(* CODESYS project WagoApp_1.11.0.x_Cloud_FbCollectionLogger_Example_03.ecp

Project tree, tasks and I/O mapping:
  PFC_KQL : 750-8210 PFC200 G2 4ETH, WAGO, order no. 0750-8210, version 5.17.3.3
    application Application
      libraries: ; WagoAppCloud, * (WAGO); WagoAppTime, 1.7.3.5 (WAGO); WagoAppControlSuite, 1.0.2.0 (WAGO)
      task PLC_Task (cyclic, interval 50 ms, priority 14) calls Prg_To_Cloud
      program Prg_To_Cloud [ST]
      trace Trace (task PLC_Task): Prg_To_Cloud.rSineP, Prg_To_Cloud.rValue
      FbOnChange/
        function block FbChangeOfValue_Bool [ST]
        function block FbChangeOfValue_Byte [ST]
        function block FbChangeOfValue_Dword [ST]
        function block FbChangeOfValue_Real [ST]
    ProjectConfiguration
    Kbus : Kbus, WAGO, version 1.4.0.2
        unmapped channels: K-BUS diagnostics
      _16_DO_Generic : 075x-16DO, WAGO, order no. 075x-16DO, version 0.0.0.13
          settings: K-BUS Module slot index = 3
          output wOut : WORD  // _OUT
      _2_DO_Generic : 075x-2DO, WAGO, order no. 075x-2DO, version 0.0.0.13
          settings: K-BUS Module slot index = 1
          output xCloudConnected : BOOL  // _OUT._OUT
          output xCloudError : BOOL  // _OUT._OUT
          unmapped channels: _OUT
      _16_DI_Generic : 075x-16DI, WAGO, order no. 075x-16DI, version 0.0.0.13
          settings: K-BUS Module slot index = 2
          input  wIn : WORD  // _IN
      _2AI_0_10_VDC_SE : 0750-0467, WAGO, order no. 0750-0467, version 0.0.0.9
          settings: K-BUS Module slot index = 4
          input  wAnalog_0_10V_1 : WORD  // _IW 1
          input  wAnalog_0_10V_2 : WORD  // _IW 2
      _2AI_TC_K_Diagn_Adjust : 0750-0469/0003-0000, WAGO, order no. 0750-0469/0003-0000, version 0.0.0.9
          settings: K-BUS Module slot index = 5
          input  iThermo1 : INT  // _IINT 1
          input  iThermo2 : INT  // _IINT 2
      _2AO_0_10_VDC : 0750-0550, WAGO, order no. 0750-0550, version 0.0.0.9
          settings: K-BUS Module slot index = 6
          output wAnalogOut_0_10V_1 : WORD  // _QW 1
          output wAnalogOut_0_10V_2 : WORD  // _QW 2
    MODBUS
      MODBUS : MODBUS, WAGO, order no. n/a, version 1.1.1.16
    Common.PCI
    EtherNet/IP
      Ethernet : Ethernet, WAGO, version 35.17.0.0
          settings: IPAddress = [192, 168, 1, 103]; SubnetMask = [0, 0, 0, 0]; MACAddress = [16#00, 16#00, 16#00, 16#00, 16#00, 16#00]; NetworkInterfaceName = 'br0'; NetworkInterfaceName = "br0"
  EC_PIO3_C : Edge Controller PIO3, WAGO, order no. 0752-8303, version 5.17.3.3
    application Application
      libraries: ; WagoAppTime, 1.7.3.5 (WAGO)
      task PLC_Task (cyclic, interval t#50ms, priority 15) calls PLC_PRG
      program PLC_PRG [ST]
    MODBUS
      MODBUS : MODBUS, WAGO, order no. n/a, version 1.1.1.16
    CANbus
    TP600_Onboard_IO : TP600 Onboard IO, WAGO, version 0.0.1.2
        output bOut : BYTE  // _OUT
        unmapped channels: _IN
    Common.PCI
    EtherNet/IP
      Ethernet : Ethernet, WAGO, version 35.17.0.0
          settings: IPAddress = [192, 168, 1, 14]; SubnetMask = [0, 0, 0, 0]; MACAddress = [16#00, 16#00, 16#00, 16#00, 16#00, 16#00]; NetworkInterfaceName = 'br0'; NetworkInterfaceName = "br0"
    Serial
      COM1 : COM1, WAGO, version 0.0.0.19
  00000000-0000-0000-0000-000000000000|C:\Users\Admin\AppData\Local\Temp\6c95a57c3216420fa36a3ac6dc2d92b7\e868b832187f4f1a859da50215710801\20221104120952\Project.xml
*)

// PFC_KQL/Application/Prg_To_Cloud
(* Purpose of the example program: 
	FbCollectionLogger will sample 3 collections in different modes.
	- Collection 1: EQUALLY_SPACED_COLLECTION_SAMPLES
	- Collection 2: UNEQUALLY_SPACED_CUSTOMIZED_SAMPLES
	- Collection 3: LIBRARY_DEFAULT_AUTOMATIC
*)
PROGRAM Prg_To_Cloud
VAR RETAIN
	(* Remanent variables *)
	tSampleInterval1 : TIME := T#10s;
	tPublishInterval1 : TIME := T#20S;
	tPublishInterval2 : TIME := T#20S;
	tSampleInterval3 : TIME := T#60S;
	tPublishInterval3 : TIME := T#120S;
xEnablePID: BOOL;rKp: REAL := 1.4;rTn: REAL := 19.89;rTv: REAL := 0.021;END_VAR

VAR
	

	(* Define three collections*)
	aCollections: ARRAY[0..2] OF WagoAppCloud.typCollection;

	(* Define the variables for the collections*)
	aVariableDescriptions1: ARRAY[0..3] OF WagoAppCloud.typVariableDescription;
	aVariableDescriptions2: ARRAY[0..2] OF WagoAppCloud.typVariableDescription;
	aVariableDescriptions3: ARRAY[0..5] OF WagoAppCloud.typVariableDescription;
	
	oFbCollectionLogger: WagoAppCloud.FbCollectionLogger;
	
	(* Timer *)
	xEnableTimer: BOOL := TRUE;
	tCyclicTimerSendTagCollection: TON;

	oFbChangeOfValue_Dword: FbChangeOfValue_Dword;	
	
	rPercentage1: REAL;
	rPercentage2: REAL;
	rTemperature1: REAL;
	rTemperature2: REAL;

	oFbChangeOfValue: FbChangeOfValue_Bool;
	xInputChanged: BOOL;
	xOutputChanged: BOOL;
	x: REAL := 0.01;
	wValue: WORD;
	rSineP: REAL;
	rValue: REAL;
	oFbStatus_WagoProtocol: WagoAppCloud.FbStatus_WagoProtocol;
	rCache: REAL;
	tSampleInterval1_10Minute: TIME := t#10m;
	xOutSend: BOOL;
	oFbChangeOfValue2: FbChangeOfValue_Bool;
	typComp: WagoAppTime.WagoTypes.typWagoTimeComponents;
	oRT: R_TRIG;
	
	oFb_PID_01: WagoAppControlSuite.Fb_PID_01;
	
	rSetpointTemperature1: REAL := 36.4;
	tSampleRate: TIME := T#100ms;
	
	
	
	rOutputMax: REAL := 100;
	rOutputMin: REAL := 0;
	xManualOperation: BOOL;
	rManualValue: REAL := 42.42;
	typConfiguration: WagoAppControlSuite.typPID_Configuration;
	rY: REAL;
	xLimitReached: BOOL;
	xLimitMaxReached: BOOL;
	xLimitMinReached: BOOL;
	tPublishInterval_USCD: TIME := T#10m;
	oFbChangeOfValue_Real: ARRAY[1..4] OF FbChangeOfValue_Real;
	oFbChangeOfValue_Bool_PID1,oFbChangeOfValue_Bool_PID2 :FbChangeOfValue_Bool;
END_VAR


typComp:=WagoAppTime.FuGetLocalTimeComponents();
oRT(CLK:=typComp.uiSecond.0);
IF oRT.Q THEN
	
	
	rPercentage1:= IoConfig_Globals_Mapping.wAnalog_0_10V_1/327.6;
	rPercentage2:= IoConfig_Globals_Mapping.wAnalog_0_10V_2/327.6;
	
	rTemperature1:= IoConfig_Globals_Mapping.iThermo1/10.0;
	rTemperature2:= IoConfig_Globals_Mapping.iThermo2/10.0;
	
	IF x > 3.14 THEN
		x:=0;
		ELSE 
			x:=x+0.01;	
	END_IF
	rSineP:=SIN(x);
	rValue:=rSineP * 32760;
	wValue:=TO_WORD(rValue);
END_IF

oFb_PID_01(
	xEnable:= 		xEnablePID, 
	rActualValue:=	rTemperature1 , 
	rSetpointValue:=rSetpointTemperature1 , 
	tSampleRate:= 	tSampleRate, 
	rKp:=	rKp , 
	rTn:= 	rTn, 
	rTv:=	rTv , 
	rOutputMax:=		rOutputMax, 
	rOutputMin:=		rOutputMin , 
	xManualOperation:= xManualOperation, 
	rManualValue:= 		rManualValue, 
	typConfiguration:= 	typConfiguration, 
	rY=> rY, 
	xLimitReached=>   xLimitReached , 
	xLimitMaxReached=>xLimitMaxReached , 
	xLimitMinReached=>xLimitMinReached);
//Generate some values for AO and DO	
IoConfig_Globals_Mapping.wAnalogOut_0_10V_1:= wValue;
IoConfig_Globals_Mapping.wOut:=(IoConfig_Globals_Mapping.wAnalog_0_10V_1 + IoConfig_Globals_Mapping.wAnalog_0_10V_2)/2;

(* Configuration of the collections and variables *)
	(* Init collection 1 *)
	aVariableDescriptions1[0].pAddress := ADR(rPercentage1);
	aVariableDescriptions1[0].eValueType := WagoAppCloud.VVT_REAL;
	aVariableDescriptions1[0].dwTypeId := 1;
	aVariableDescriptions1[0].sTag := 'Inflow1';
	aVariableDescriptions1[0].sUnit := '';
	
	aVariableDescriptions1[1].pAddress := ADR(rPercentage2);
	aVariableDescriptions1[1].eValueType := WagoAppCloud.VVT_REAL;
	aVariableDescriptions1[1].dwTypeId := 2;
	aVariableDescriptions1[1].sTag := 'Inflow2';
	aVariableDescriptions1[1].sUnit := '';
	
	aVariableDescriptions1[2].pAddress := ADR(rTemperature1);
	aVariableDescriptions1[2].eValueType := WagoAppCloud.VVT_REAL;
	aVariableDescriptions1[2].dwTypeId := 3;
	aVariableDescriptions1[2].sTag := 'Temperature1';
	aVariableDescriptions1[2].sUnit := '°C';
	
	aVariableDescriptions1[3].pAddress := ADR(rTemperature2);
	aVariableDescriptions1[3].eValueType := WagoAppCloud.VVT_REAL;
	aVariableDescriptions1[3].dwTypeId := 4;
	aVariableDescriptions1[3].sTag := 'Temperature2';
	aVariableDescriptions1[3].sUnit := '°C';
	
	
	(* Configuration of the collection. *)
	aCollections[0].dwCollectionId := 1;
	aCollections[0].sName := 'CollectionAnalogs';
	aCollections[0].pVariableDescriptions := ADR(aVariableDescriptions1);
	aCollections[0].dwVariablesCount := 4;
	(* Configuration of the mode to sampling the data. 
	In this case all variables of collection 1 will be send in equally spaced to the cloud. 
	The Trigger of a sample is set manual with the CollectionTrigger. *)
	aCollections[0].eSamplingDataMode := eSamplingMode.LIBRARY_DEFAULT_AUTOMATIC;
	aCollections[0].pSampleInterval := ADR(tSampleInterval1);
	aCollections[0].pPublishInterval := ADR(tPublishInterval1);
	
	(* Init collection 2 *)
	aVariableDescriptions2[0].pAddress := ADR(IoConfig_Globals_Mapping.wIn);
	aVariableDescriptions2[0].eValueType := WagoAppCloud.VVT_WORD;
	aVariableDescriptions2[0].dwTypeId := 1;
	aVariableDescriptions2[0].sTag := 'DI';
	aVariableDescriptions2[0].sUnit := 'Bin';
	
	aVariableDescriptions2[1].pAddress := ADR(IoConfig_Globals_Mapping.wOut);
	aVariableDescriptions2[1].eValueType := WagoAppCloud.VVT_WORD;
	aVariableDescriptions2[1].dwTypeId := 2;
	aVariableDescriptions2[1].sTag := 'DO';
	aVariableDescriptions2[1].sUnit := 'Bin';
	
	
	(* Configuration of the collection. *)
	aCollections[1].dwCollectionId := 2;
	aCollections[1].sName := 'CollectionDigital';
	aCollections[1].pVariableDescriptions := ADR(aVariableDescriptions2);
	aCollections[1].dwVariablesCount := 2;
	(* Configuration of the mode to sampling the data. 
	In this case at least one variable of collection 2 will be send irregularly to the cloud. 
	The Trigger of a sample is set manual with the CollectionTrigger or the VariableTrigger. *)
	aCollections[1].eSamplingDataMode := eSamplingMode.EQUALLY_SPACED_CUSTOMIZED_SAMPLES;
	aCollections[1].pPublishInterval := ADR(tPublishInterval2);
	(* Configuration of the collection. *)
	
	
	aVariableDescriptions3[0].pAddress := ADR(xEnablePID);
	aVariableDescriptions3[0].eValueType := WagoAppCloud.VVT_BOOL;
	aVariableDescriptions3[0].dwTypeId := 1;
	aVariableDescriptions3[0].sTag := 'EN';
	aVariableDescriptions3[0].sUnit := 'Bin';
	                     
	aVariableDescriptions3[1].pAddress := ADR(rSetpointTemperature1);
	aVariableDescriptions3[1].eValueType := WagoAppCloud.VVT_REAL;
	aVariableDescriptions3[1].dwTypeId := 2;
	aVariableDescriptions3[1].sTag := 'Setpoint';
	aVariableDescriptions3[1].sUnit := '°C';
	
	aVariableDescriptions3[2].pAddress := ADR(rKp);
	aVariableDescriptions3[2].eValueType := WagoAppCloud.VVT_REAL;
	aVariableDescriptions3[2].dwTypeId := 3;
	aVariableDescriptions3[2].sTag := 'P';
	aVariableDescriptions3[2].sUnit := '';
	                     
	aVariableDescriptions3[3].pAddress := ADR(rTn);
	aVariableDescriptions3[3].eValueType := WagoAppCloud.VVT_REAL;
	aVariableDescriptions3[3].dwTypeId := 4;
	aVariableDescriptions3[3].sTag := 'I';
	aVariableDescriptions3[3].sUnit := '';
	
	aVariableDescriptions3[4].pAddress := ADR(rTv);
	aVariableDescriptions3[4].eValueType := WagoAppCloud.VVT_REAL;
	aVariableDescriptions3[4].dwTypeId := 5;
	aVariableDescriptions3[4].sTag := 'D';
	aVariableDescriptions3[4].sUnit := '';
	                     
	aVariableDescriptions3[5].pAddress := ADR(xManualOperation);
	aVariableDescriptions3[5].eValueType := WagoAppCloud.VVT_BOOL;
	aVariableDescriptions3[5].dwTypeId := 6;
	aVariableDescriptions3[5].sTag := 'ManuelOperation';
	aVariableDescriptions3[5].sUnit := 'Bin';
	
	aCollections[2].dwCollectionId := 3;
	aCollections[2].sName := 'CollectionPID';
	aCollections[2].pVariableDescriptions := ADR(aVariableDescriptions3);
	aCollections[2].dwVariablesCount := 6;
	aCollections[2].eSamplingDataMode := eSamplingMode.UNEQUALLY_SPACED_CUSTOMIZED_SAMPLES;
	aCollections[2].pPublishInterval := ADR(tPublishInterval_USCD);
	
	
		
// BOOL on change
oFbChangeOfValue_Bool_PID1(xVariable:=xEnablePID 		, xTrigger:= aVariableDescriptions3[0].xVariableTrigger);
oFbChangeOfValue_Bool_PID2(xVariable:=xManualOperation  , xTrigger:= aVariableDescriptions3[5].xVariableTrigger);
 //xEnable PID Controller
 //Manuel Operation


// REAL  on change	
oFbChangeOfValue_Real[1](rInput:=rSetpointTemperature1 ,
						 rActivate:= 100 , 
						 rDeactivate:= 0, 							xTrigger:=aVariableDescriptions3[1].xVariableTrigger);
						 
oFbChangeOfValue_Real[2](rInput:=rKp , rActivate:=0 , rDeactivate:=100, xTrigger:=aVariableDescriptions3[2].xVariableTrigger);
oFbChangeOfValue_Real[3](rInput:=rTn , rActivate:=0 , rDeactivate:=100 ,xTrigger:=aVariableDescriptions3[3].xVariableTrigger);
oFbChangeOfValue_Real[4](rInput:=rTv , rActivate:=0 , rDeactivate:=100 ,xTrigger:=aVariableDescriptions3[4].xVariableTrigger);






(* Example to set the event if variable value exceeded the threshold values - Variable Trigger*)

oFbChangeOfValue(xVariable:=	wIn.0 OR 
								wIn.1 OR 
								wIn.2 OR 
								wIn.3 OR 
								wIn.4 OR 
								wIn.5 OR 
								wIn.6 OR 
								wIn.7, 
					xTrigger:= aVariableDescriptions2[0].xVariableTrigger);
	
oFbChangeOfValue2(xVariable:=	wOut.0 OR 
								wOut.1 OR 
								wOut.2 OR 
								wOut.3 OR 
								wOut.4 OR 
								wOut.5 OR 
								wOut.6 OR 
								wOut.7, 
					xTrigger:= aVariableDescriptions2[1].xVariableTrigger);

	
	

(* Example to set the event with a timer intervall - CollectionTrigger or VariableTrigger *)
	(* Set an event with an Timer to send the variables in an intervall to the cloud *)
	tCyclicTimerSendTagCollection(IN:= xEnableTimer, PT:= tSampleInterval1_10Minute);
	IF tCyclicTimerSendTagCollection.Q THEN
		aCollections[1].xCollectionTrigger := TRUE;
		aCollections[2].xCollectionTrigger:=TRUE;
		xEnableTimer := FALSE;
	ELSE
		xEnableTimer := TRUE;
	END_IF

	
oFbCollectionLogger(pCollections := ADR(aCollections), dwCollectionsCount := 3);
oFbStatus_WagoProtocol(
	xEnabled:=TRUE , 
	xError=>IoConfig_Globals_Mapping.xCloudError , 
	xCloudConnected=> IoConfig_Globals_Mapping.xCloudConnected, 
	rCacheFillLevel=> rCache , 
	xTelemetryDataTransmission=> , 
	bCollectionCounter=> , 
	uliOutgoingDataBlocks=> , 
	ErrorInformation=> , 
	oStatus=> );

END_PROGRAM

// PFC_KQL/Application/FbOnChange/FbChangeOfValue_Dword
(* The function block FbChangeOfValue_Dword shows an example how an event of a dword variable could be triggered.*)

FUNCTION_BLOCK FbChangeOfValue_Dword

VAR_INPUT
	dwInput 	: DWORD;
	dwActivate 	: DWORD;
	dwDeactivate : DWORD;
END_VAR

VAR_IN_OUT
	xTrigger	: BOOL;
END_VAR

VAR
	xLastSendedState: BOOL := FALSE;
END_VAR

(* Do only something when the VariableTrigger isn't activated (the VariableTrigger will be reset by the function block FbCollectionLogger) *)
IF NOT xTrigger THEN
	(* Two variations are to be considered during the analysis of the input values *)
	
	(* case 1: the activate threshold is greater as the deactivate threshold *)	
	IF dwActivate > dwDeactivate THEN
		(* rising edge *)
		IF (dwInput >= dwActivate) AND NOT xLastSendedState THEN
			xTrigger := TRUE;
			xLastSendedState := TRUE;
		(* falling edge *)
		ELSIF (dwInput <= dwDeactivate) AND xLastSendedState THEN
			xTrigger := TRUE;
			xLastSendedState := FALSE;
		END_IF
		
	(* case 2: the deactivate threshold is greater as the activate threshold *)
	ELSE
		(* rising edge *)
		IF (dwInput <= dwActivate) AND NOT xLastSendedState THEN
			xTrigger := TRUE;
			xLastSendedState := TRUE;(* save that the trigger after the rising edge is already set so that the trigger will be only set once *)
		(* falling edge *)
		ELSIF (dwInput >= dwDeactivate) AND xLastSendedState THEN
			xTrigger := TRUE;
			xLastSendedState := FALSE;
		END_IF
	END_IF
END_IF

END_FUNCTION_BLOCK

// PFC_KQL/Application/FbOnChange/FbChangeOfValue_Bool
FUNCTION_BLOCK FbChangeOfValue_Bool
VAR_INPUT
	xVariable : BOOL; 	(* Input value *)
END_VAR
VAR_IN_OUT
	xTrigger : BOOL; 	(* Variable Trigger - trigger is set only once when the value was changed and reset with the function block WagoAppCloud.FbCollectionLogger *)
END_VAR
VAR
	xLastSendedState : BOOL := FALSE; 	(* save the old value when this value was sending to the cloud to the if the value was changing *)
END_VAR

IF NOT xTrigger THEN
	IF NOT (xVariable = xLastSendedState) THEN
		xTrigger := TRUE;
		xLastSendedState := xVariable;
	END_IF
END_IF

END_FUNCTION_BLOCK

// PFC_KQL/Application/FbOnChange/FbChangeOfValue_Real
(* The function block FbChangeOfValue_Real shows an example how an event of a real variable could be triggered.
*)

FUNCTION_BLOCK FbChangeOfValue_Real

VAR_INPUT
	rInput 		: REAL;
	rActivate 	: REAL;
	rDeactivate : REAL;
END_VAR

VAR_IN_OUT
	xTrigger	: BOOL;
END_VAR

VAR
	xLastSendedState : BOOL := FALSE;
END_VAR

IF NOT xTrigger THEN
	IF rActivate > rDeactivate THEN
		IF (rInput >= rActivate) AND NOT xLastSendedState THEN
			xTrigger := TRUE;
			xLastSendedState := TRUE;
		ELSIF (rInput <= rDeactivate) AND xLastSendedState THEN
			xTrigger := TRUE;
			xLastSendedState := FALSE;
		END_IF
	ELSE
		IF (rInput <= rActivate) AND NOT xLastSendedState THEN
			xTrigger := TRUE;
			xLastSendedState := TRUE;
		ELSIF (rInput >= rDeactivate) AND xLastSendedState THEN
			xTrigger := TRUE;
			xLastSendedState := FALSE;
		END_IF
	END_IF
END_IF

END_FUNCTION_BLOCK

// EC_PIO3_C/Application/PLC_PRG
PROGRAM PLC_PRG
VAR
	typComp: WagoAppTime.WagoTypes.typWagoTimeComponents;
	oRT: R_TRIG;
END_VAR

typComp:=WagoAppTime.FuGetLocalTimeComponents();
oRT(CLK:=typComp.uiSecond.0);
IF oRT.Q THEN
	IF IoConfig_Globals_Mapping.bOut <=255 THEN
	IoConfig_Globals_Mapping.bOut:=IoConfig_Globals_Mapping.bOut+1;
	ELSE
		IoConfig_Globals_Mapping.bOut:=0;
	END_IF
END_IF

END_PROGRAM

// PFC_KQL/Application/FbOnChange/FbChangeOfValue_Byte
(* The function block FbChangeOfValue_Byte shows an example how an event of a real variable could be triggered.
*)

FUNCTION_BLOCK FbChangeOfValue_Byte

VAR_INPUT
	bInput 		: BYTE; (* Input value *)
	bActivate 	: BYTE; (* Threshold value at which the output signal is set to TRUE *)
	bDeactivate : BYTE; (* Threshold value at which the output signal is set to FALSE *)
END_VAR

VAR_IN_OUT
	xTrigger	: BOOL; (* VariableTrigger - trigger is set only once when the value was changed and reset with the function block WagoAppCloud.FbCollectionLogger *)
END_VAR

VAR
	xLastSendedState : BOOL := FALSE; (* state of the last sended changed state - send a change only once when the threshold was exceeded *)
END_VAR

(* Do only something when the VariableTrigger isn't activated (the VariableTrigger will be reset by the function block FbCollectionLogger) *)
IF NOT xTrigger THEN
	(* Two variations are to be considered during the analysis of the input values *)
	
	(* case 1: the activate threshold is greater as the deactivate threshold *)	
	IF bActivate > bDeactivate THEN
		(* rising edge *)
		IF (bInput >= bActivate) AND NOT xLastSendedState THEN
			xTrigger := TRUE;
			xLastSendedState := TRUE;
		(* falling edge *)
		ELSIF (bInput <= bDeactivate) AND xLastSendedState THEN
			xTrigger := TRUE;
			xLastSendedState := FALSE;
		END_IF
		
	(* case 2: the deactivate threshold is greater as the activate threshold *)
	ELSE
		(* rising edge *)
		IF (bInput <= bActivate) AND NOT xLastSendedState THEN
			xTrigger := TRUE;
			xLastSendedState := TRUE; (* save that the trigger after the rising edge is already set so that the trigger will be only set once *)
		(* falling edge *)
		ELSIF (bInput >= bDeactivate) AND xLastSendedState THEN
			xTrigger := TRUE;
			xLastSendedState := FALSE;
		END_IF
	END_IF
END_IF

END_FUNCTION_BLOCK
